// Mitsubishi GX Works2 project: e099   PLC: Q02/Q02H

PROGRAM MAIN
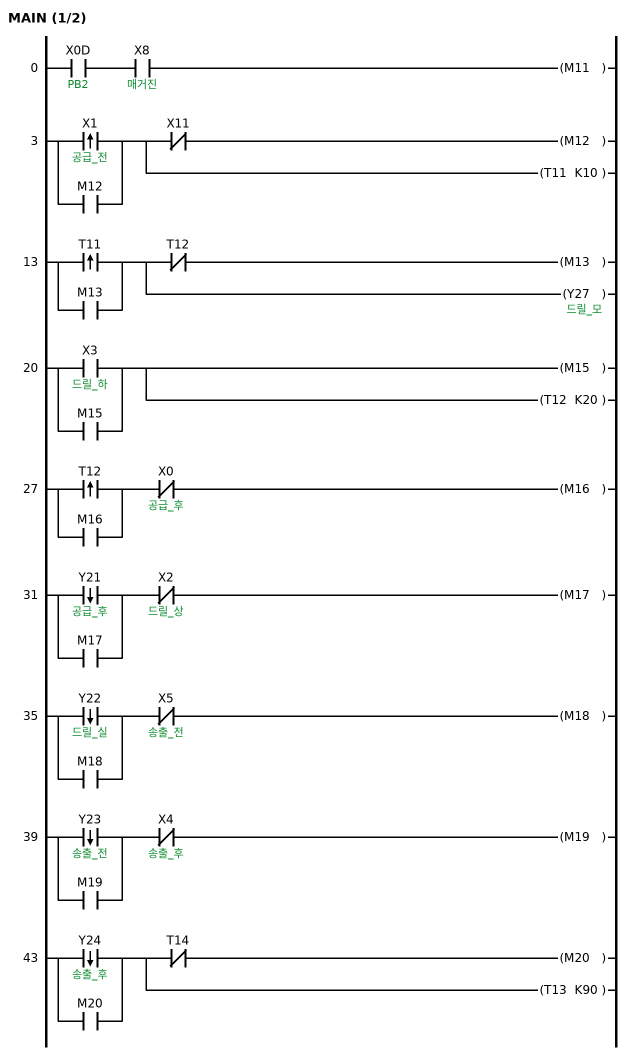
0     LD      X0D  ; PB2
      AND     X8  ; 매거진
      OUT     M11
3     LDP     X1  ; 공급_전
      OR      M12
      MPS
      ANI     X11
      OUT     M12
      MPP
      OUT     T11 K10
13    LDP     T11
      OR      M13
      MPS
      ANI     T12
      OUT     M13
      MPP
      OUT     Y27  ; 드릴_모
20    LD      X3  ; 드릴_하
      OR      M15
      OUT     M15
      OUT     T12 K20
27    LDP     T12
      OR      M16
      ANI     X0  ; 공급_후
      OUT     M16
31    LDF     Y21  ; 공급_후
      OR      M17
      ANI     X2  ; 드릴_상
      OUT     M17
35    LDF     Y22  ; 드릴_실
      OR      M18
      ANI     X5  ; 송출_전
      OUT     M18
39    LDF     Y23  ; 송출_전
      OR      M19
      ANI     X4  ; 송출_후
      OUT     M19
43    LDF     Y24  ; 송출_후
      OR      M20
      MPS
      ANI     T14
      OUT     M20
      MPP
      OUT     T13 K90
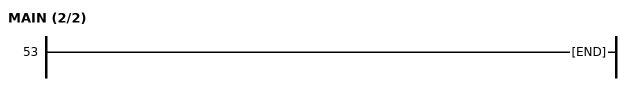
53    END
END_PROGRAM

// device comments not shown above
X6  ; 배출_후
X7  ; 배출_전
X9  ; 이송감지
X0A  ; 비금속
X0B  ; 금속
X0C  ; PB1
X0E  ; PB3
X0F  ; 비상정지
Y20  ; 공급_전
Y25  ; 배출_전
Y26  ; 배출_후
Y28  ; 컨베
Y29  ; 적램
Y2A  ; 황램
Y2B  ; 녹램
